// TwinCAT 3 PLC project main
// ProgramVersion: 3.1.4023.0
// libraries:
//   Tc2_Standard, * (Beckhoff Automation GmbH)
//   Tc2_System, * (Beckhoff Automation GmbH)
//   Tc3_Module, * (Beckhoff Automation GmbH)
// project tree:
//   DUTs/ State.TcDUT, StateCnv.TcDUT (not stored), StateDisp.TcDUT, StateHeat.TcDUT (not stored), StateMan.TcDUT (not stored), StateSeparator.TcDUT (not stored), StateTr.TcDUT (not stored), StateVe.TcDUT (not stored)
//   GVLs/ AdsVariables.TcGVL, CodeGeneration.TcGVL, IFC_HW.TcGVL
//   / PlcTask.TcTTO (not stored)
//   POUs/ FB_Conveyor.TcPOU (not stored), FB_Dispenser.TcPOU (not stored), FB_FillLevel.TcPOU (not stored), FB_HeatingSystem.TcPOU (not stored), FB_ManipulatorAxis.TcPOU (not stored), FB_RFID.TcPOU (not stored), FB_Separator.TcPOU (not stored), FB_StatusLight.TcPOU (not stored), FB_Transport.TcPOU (not stored), FB_Waage.TcPOU (not stored), MAIN.TcPOU
//   POUs/Modelle/ Model_Seperator.TcPOU (not stored)

// ---- DUTs/State.TcDUT
{attribute 'qualified_only'}
{attribute 'strict'}
TYPE State :
(
	Off,
	Busy,
	Ready,
	Done,
	Error,
	Setup
);
END_TYPE

// ---- DUTs/StateDisp.TcDUT
{attribute 'qualified_only'}
{attribute 'strict'}
TYPE StateDisp :
(
	Off := 0,
	Reset,
	PowerUp,
	Idle,
	Dispensing,
	Done
);
END_TYPE

// ---- GVLs/AdsVariables.TcGVL
{attribute 'qualified_only'}
VAR_GLOBAL
	VonMatlab		: REAL := 1;
	NachMatlab		: REAL := 1;
END_VAR

// ---- GVLs/CodeGeneration.TcGVL
VAR_GLOBAL CONSTANT
	SS_INITIALIZE: SINT := 0;
	SS_STEP: SINT := 1;
END_VAR

// ---- GVLs/IFC_HW.TcGVL
// In dieser GVL werden alle Variablen deklariert die auf die realen Klemmen zugreifen
VAR_GLOBAL

		isSimulation		: BOOL := TRUE;	

	// Errors 
		NoBottle			: BOOL := FALSE; // Keine Flasche vorhanden
		WrongBottle			: BOOL := FALSE; // Flasche falsch gedreht oder falsche Flasche
		StorageFull			: BOOL := FALSE; // Lager abgefüllte Flaschen voll
		GranulateEmpty		: BOOL := FALSE; // Füllstand Granulat zu gering
		
	// Station Statusampel	
		AmpelRot 	AT%Q* 	: BOOL;		// Signal-LED Rot
		AmpelGelb 	AT%Q* 	: BOOL;		// Signal-LED Gelb
		AmpelGrun 	AT%Q* 	: BOOL;		// Signal-LED Grun
			
	// Station Vereinzelung
		EinzelSens1 AT%I*	: BOOL;			// Separation Sensor 1
		EinzelSens2 AT%I*	: BOOL;			// Separation Sensor 2
		EinzelSens3 AT%I*	: BOOL;			// Separation Sensor 3
		R1AKT1 	AT%Q* 		: BOOL;			// Relais 1 Aktor 1
		R2AKT1 	AT%Q* 		: BOOL;			// Relais 2 Aktor 1
		R1AKT2 	AT%Q* 		: BOOL;			// Relais 1 Aktor 2
		R2AKT2 	AT%Q* 		: BOOL;			// Relais 2 Aktor 2
	
	// Station Forderband
		BandSens1 AT %I*	: BOOL;		// Forderband Sensor 1
		BandSens2 AT %I*	: BOOL;		// Forderband Sensor 2
		BandSens3 AT %I*	: BOOL;		// Forderband Sensor 3
		BandSens4 AT %I*	: BOOL;		// Forderband Sensor 4
		BandHub1 AT %Q*		: BOOL;		// Forderband Hubmagnet 1
		BandHub2 AT %Q*		: BOOL;		// Forderband Hubmagnet 1
		BandHub3 AT %Q*		: BOOL;		// Forderband Hubmagnet 1
//		BandExtruder1 		: AXIS_REF;	// Forderband NC-Achse Dosiereinheit 1
//		BandExtruder2 		: AXIS_REF;	// Forderband NC-Achse Dosiereinheit 2
//		BandExtruder3 		: AXIS_REF;	// Forderband NC-Achse Dosiereinheit 3
//		BandMotor 			: AXIS_REF;	// Forderband NC-Achse Band
		
		BandFullmenge1		: INT := 5;	// in Gramm
		BandFullmenge2		: INT := 7;	// in Gramm
		BandFullmenge3		: INT := 3;	// in Gramm
		
	//Füllstandsüberwachung
		FillSens1 AT%I*	: UINT;			// Füllstandssensor 1
		FillSens2 AT%I*	: UINT;			// Füllstandssensor 2
		FillSens3 AT%I*	: UINT;			// Füllstandssensor 3
		FillLevelPercent1	: REAL;		// Füllstand 1 in %
		FillLevelGramm1		: REAL;		// Füllstand i in g
		FillLevelPercent2	: REAL;		// Füllstand 2 in %
		FillLevelGramm2		: REAL;		// Füllstand 2 in g
		FillLevelPercent3	: REAL;		// Füllstand 3 in %
		FillLevelGramm3		: REAL;		// Füllstand 3 in g
		
		MaxFillLevel 	: REAL := 375;	// Kalibrierter Füllstand für 10% * 10
		
	// Station Waage
		WaageNachricht		: STRING;	// Nachricht von Wagezelle (fur virtuelle Inbetriebnahme notig)
		WaageNull			: BOOL;		// TARA Waage
		WaageMesswert		: INT;		// Messwert der Waage
		
	// Station Behalteridentifikation
		IdSensorTrager			: BOOL;		// Sensor bei Erkennung eines Datentrager
		IdNachricht				: STRING;	// Nachricht von RFID-System (fur virtuelle Inbetriebnahme notig)
		Seriennummer			: STRING;	// Seriennummer RFID-Tag
		
	//Temperierstation
		Ventilator1 AT %Q*	: BOOL;		// Ventilator 1
		Ventilator2 AT %Q*	: BOOL;		// Ventilator 2
		Ventilator3 AT %Q*	: BOOL;		// Ventilator 3
		TempSens1 AT%I*		: UINT;		// Temperatursensor 1
		TempSens2 AT%I*		: UINT;		// Temperatursensor 2
		Heizpatrone AT%Q*	: UINT;		// Heizpatronen
		MaxTemp				: UINT := 5500;		// in °C * 100
		
	// Station Manipulator
		ManEndX AT%I* 		: BOOL := TRUE;		// Manipulator min Endschalter Achse x
		ManEndY AT%I* 		: BOOL := TRUE;		// Manipulator min Endschalter Achse y
		ManEndZ AT%I* 		: BOOL := TRUE;		// Manipulator min Endschalter Achse z
		ManEndGrip AT%I* 	: BOOL := TRUE;		// Manipulator min Endschalter Achse Gripper
		ManEndX2 AT%I* 		: BOOL := TRUE;		// Manipulator max Endschalter Achse x
		ManEndY2 AT%I* 		: BOOL := TRUE;		// Manipulator max Endschalter Achse y
		ManEndZ2 AT%I* 		: BOOL := TRUE;		// Manipulator max Endschalter Achse z
		ManEndGrip2 AT%I* 	: BOOL := TRUE;		// Manipulator max Endschalter Achse Gripper
		Brake	AT%Q*		: BOOL := FALSE;	// Bremse Achse z
		
//		ManAchseX			: AXIS_REF;			// Manipulator NC-Achse x
//		ManAchseY			: AXIS_REF;			// Manipulator NC-Achse y
//		ManAchseZ			: AXIS_REF;			// Manipulator NC-Achse z
//		ManAchseGrip		: AXIS_REF; 		// Manipulator NC-Achse Gripper

// Visualization Inventor
	Inv_Vereinz_Container1  :  	REAL := 0;
    Inv_Vereinz_Container2  :  	REAL := 0;
    Inv_Vereinz_Container3  :  	REAL := 0;
    Inv_Vereinz_Container4  :  	REAL := 0;
    Inv_Vereinz_Container5  :  	REAL := 0;
	
	Inv_Vereinz_HubmagnetOben	: 	REAL := 0;
	Inv_Vereinz_HubmagnetUnten	:	REAL := 0;

END_VAR

// ---- POUs/MAIN.TcPOU
PROGRAM MAIN
VAR
	iState 		: INT 	:= 0;	
	iMethod		: SINT 	:= 0;
	
	bCreateContainer	: 	BOOL := FALSE;
	bRemoveContainer	:	BOOL := FALSE;
	
	
	bSensorLagerUnten		: BOOL;
	bSensorLagerMitte		: BOOL; 
	
	
	fbSeperator		: FB_Separator;
	staSep			: State;
	instVereinzelung : Model_Seperator;
	
	temp	: BOOL := FALSE;
	enzSens1 : BOOL;
	enzSens2 : BOOL;
	enzSens3 : BOOL;
END_VAR

IF(IFC_HW.isSimulation = TRUE) THEN
	// Call models	
instVereinzelung(
	ssMethodType:= iMethod, Signal_CreateContainer:= bCreateContainer, 	c_Signal_RemoveContainerOnC:= bRemoveContainer, 
	SamplingTime:= 0.005, 
	Hw_AktObenEinfahren:= IFC_HW.R1AKT1,	// einfahren
 	Hw_AktObenAusfahren:= IFC_HW.R2AKT1,	// ausfahren
	Hw_AktUntenEinfahren:= IFC_HW.R2AKT2,	// einfahren
 	Hw_AktUntenAusfahren:= IFC_HW.R1AKT2, 	// ausfahren
	Signal_Storage2=> bSensorLagerMitte,
 	Signal_Storage1=> bSensorLagerUnten, 
	Hw_SensorOben=> enzSens3,
 	Hw_SensorMitte=> enzSens2,
 	Hw_SensorUnten=> enzSens1);
IFC_HW.EinzelSens1 := enzSens1;
IFC_HW.EinzelSens2 := enzSens2;
IFC_HW.EinzelSens3 := enzSens3;

END_IF



	
// Call Functionblocks
fbSeperator(
	bEnable:= TRUE, bExecute:= temp, bErrorReset:= , 
	bSensor1:= IFC_HW.EinzelSens1,
 	bSensor2:= IFC_HW.EinzelSens2,
 	bSensor3:= IFC_HW.EinzelSens3, 
	bR1AKT1=> IFC_HW.R1AKT1,	// einfahren
 	bR2AKT1=> IFC_HW.R2AKT1,	// ausfahren
 	bR1AKT2=> IFC_HW.R1AKT2,	// ausfahren
 	bR2AKT2=> IFC_HW.R2AKT2, 	// einfahren
	bNoBottle=> IFC_HW.NoBottle, 
	bWrongBottle=> IFC_HW.WrongBottle, 
	eStatus=> staSep);	

	
// Visualization Inventor
IFC_HW.Inv_Vereinz_Container1 := BOOL_TO_REAL(IFC_HW.EinzelSens1);
IFC_HW.Inv_Vereinz_Container2 := BOOL_TO_REAL(IFC_HW.EinzelSens2);
IFC_HW.Inv_Vereinz_Container3 := BOOL_TO_REAL(IFC_HW.EinzelSens3);
IFC_HW.Inv_Vereinz_Container4 := BOOL_TO_REAL(bSensorLagerUnten);
IFC_HW.Inv_Vereinz_Container5 := BOOL_TO_REAL(bSensorLagerMitte);

IF (IFC_HW.R1AKT1 = TRUE) THEN 
	IFC_HW.Inv_Vereinz_HubmagnetOben := 1;
ELSIF (IFC_HW.R2AKT1 = TRUE) THEN
	IFC_HW.Inv_Vereinz_HubmagnetOben := 0;
END_IF

IF (IFC_HW.R2AKT2 = TRUE) THEN
	IFC_HW.Inv_Vereinz_HubmagnetUnten := 1;
ELSIF (IFC_HW.R1AKT2 = TRUE) THEN
	IFC_HW.Inv_Vereinz_HubmagnetUnten := 0;
END_IF



//AdsVariables.HubmagnetOben_ADS := BOOL_TO_REAL(bHubmagnetOben);
//AdsVariables.HubmagnetUnten_ADS := BOOL_TO_REAL(bHubmagnetUnten);
	



// State Machine
CASE iState OF
	0:
		
		iState := iState +1;
	1:
		iMethod := 1;
END_CASE

END_PROGRAM
